// TIA Portal V20 export
FUNCTION_BLOCK "FC_Traffic_Lights"   // FB1, LAD
{ S7_Optimized_Access := 'TRUE' }
// stored: MemoryReserve 100, SetENOAutomatically false
   VAR
      "Timer" { S7_SetPoint := 'True'} : TON_TIME;
   END_VAR
   VAR_TEMP   // added for the SCL form of the ladder/FBD networks
      _w1 : Bool;
   END_VAR
BEGIN

REGION Network 1
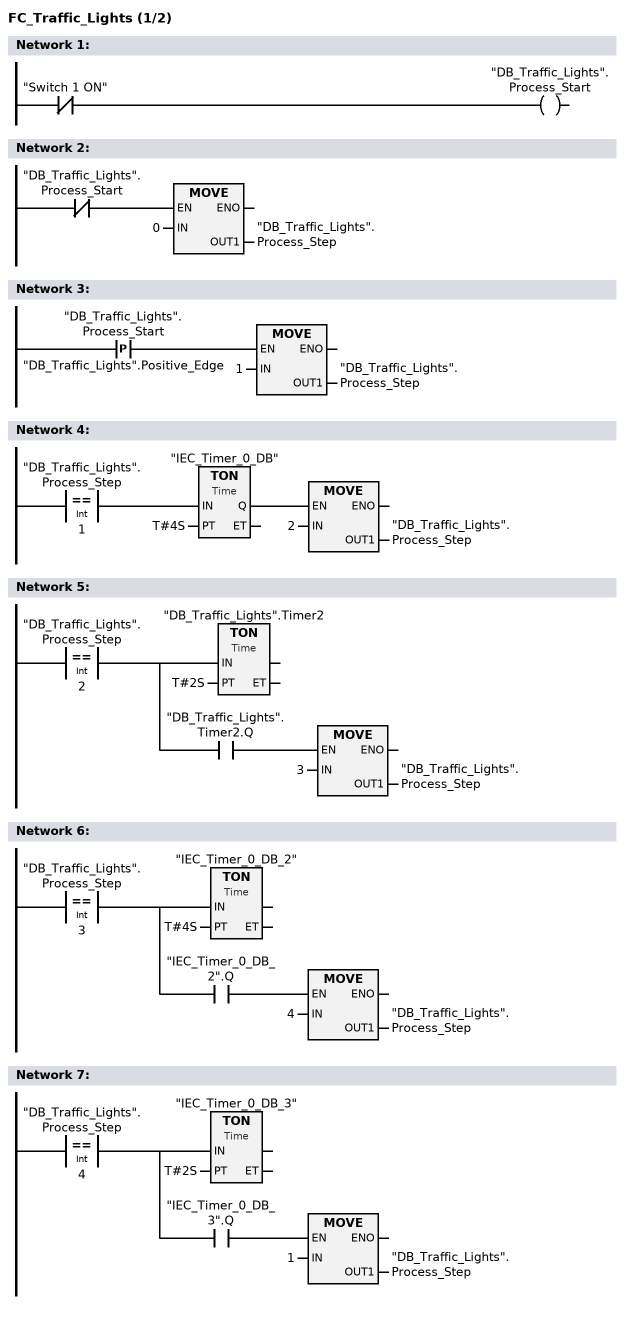
   RUNG wire#powerrail
      I_Contact( "Switch 1 ON" )
      Coil( "DB_Traffic_Lights".Process_Start )
   END_RUNG
   // the same network as SCL:
   "DB_Traffic_Lights".Process_Start := NOT "Switch 1 ON";
END_REGION

REGION Network 2
   RUNG wire#powerrail
      I_Contact( "DB_Traffic_Lights".Process_Start )
      Move(in := 0, out1 => "DB_Traffic_Lights".Process_Step)
   END_RUNG
   // the same network as SCL:
   IF NOT "DB_Traffic_Lights".Process_Start THEN "DB_Traffic_Lights".Process_Step := 0; END_IF;
END_REGION

REGION Network 3
   RUNG wire#powerrail
      P_Contact(operand := "DB_Traffic_Lights".Process_Start, bit := "DB_Traffic_Lights".Positive_Edge)
      Move(in := 1, out1 => "DB_Traffic_Lights".Process_Step)
   END_RUNG
   // the same network as SCL:
   #_w1 := "DB_Traffic_Lights".Process_Start AND NOT "DB_Traffic_Lights".Positive_Edge;   // rising edge of "DB_Traffic_Lights".Process_Start
   "DB_Traffic_Lights".Positive_Edge := "DB_Traffic_Lights".Process_Start;
   IF #_w1 THEN "DB_Traffic_Lights".Process_Step := 1; END_IF;
END_REGION

REGION Network 4
   RUNG wire#powerrail
      { S7_Templates := "SrcType := Int" } EQ_Contact(in1 := "DB_Traffic_Lights".Process_Step, in2 := 1)
      { S7_Templates := "time_type := Time" } "IEC_Timer_0_DB".TON(pt := T#4S, et =>)
      Move(in := 2, out1 => "DB_Traffic_Lights".Process_Step)
   END_RUNG
   // the same network as SCL:
   "IEC_Timer_0_DB".TON(IN := "DB_Traffic_Lights".Process_Step = 1, PT := T#4S);
   IF "IEC_Timer_0_DB".Q THEN "DB_Traffic_Lights".Process_Step := 2; END_IF;
END_REGION

REGION Network 5
   RUNG wire#powerrail
      { S7_Templates := "SrcType := Int" } EQ_Contact(in1 := "DB_Traffic_Lights".Process_Step, in2 := 2)
      wire#w1
      { S7_Templates := "time_type := Time" } "DB_Traffic_Lights".Timer2.TON(pt := T#2S, et =>)
   END_RUNG
   RUNG wire#w1
      Contact( "DB_Traffic_Lights".Timer2.Q )
      Move(in := 3, out1 => "DB_Traffic_Lights".Process_Step)
   END_RUNG
   // the same network as SCL:
   #_w1 := "DB_Traffic_Lights".Process_Step = 2;
   "DB_Traffic_Lights".Timer2.TON(IN := #_w1, PT := T#2S);
   IF #_w1 AND "DB_Traffic_Lights".Timer2.Q THEN "DB_Traffic_Lights".Process_Step := 3; END_IF;
END_REGION

REGION Network 6
   RUNG wire#powerrail
      { S7_Templates := "SrcType := Int" } EQ_Contact(in1 := "DB_Traffic_Lights".Process_Step, in2 := 3)
      wire#w1
      { S7_Templates := "time_type := Time" } "IEC_Timer_0_DB_2".TON(pt := T#4S, et =>)
   END_RUNG
   RUNG wire#w1
      Contact( "IEC_Timer_0_DB_2".Q )
      Move(in := 4, out1 => "DB_Traffic_Lights".Process_Step)
   END_RUNG
   // the same network as SCL:
   #_w1 := "DB_Traffic_Lights".Process_Step = 3;
   "IEC_Timer_0_DB_2".TON(IN := #_w1, PT := T#4S);
   IF #_w1 AND "IEC_Timer_0_DB_2".Q THEN "DB_Traffic_Lights".Process_Step := 4; END_IF;
END_REGION

REGION Network 7
   RUNG wire#powerrail
      { S7_Templates := "SrcType := Int" } EQ_Contact(in1 := "DB_Traffic_Lights".Process_Step, in2 := 4)
      wire#w1
      { S7_Templates := "time_type := Time" } "IEC_Timer_0_DB_3".TON(pt := T#2S, et =>)
   END_RUNG
   RUNG wire#w1
      Contact( "IEC_Timer_0_DB_3".Q )
      Move(in := 1, out1 => "DB_Traffic_Lights".Process_Step)
   END_RUNG
   // the same network as SCL:
   #_w1 := "DB_Traffic_Lights".Process_Step = 4;
   "IEC_Timer_0_DB_3".TON(IN := #_w1, PT := T#2S);
   IF #_w1 AND "IEC_Timer_0_DB_3".Q THEN "DB_Traffic_Lights".Process_Step := 1; END_IF;
END_REGION

REGION Network 8: Step
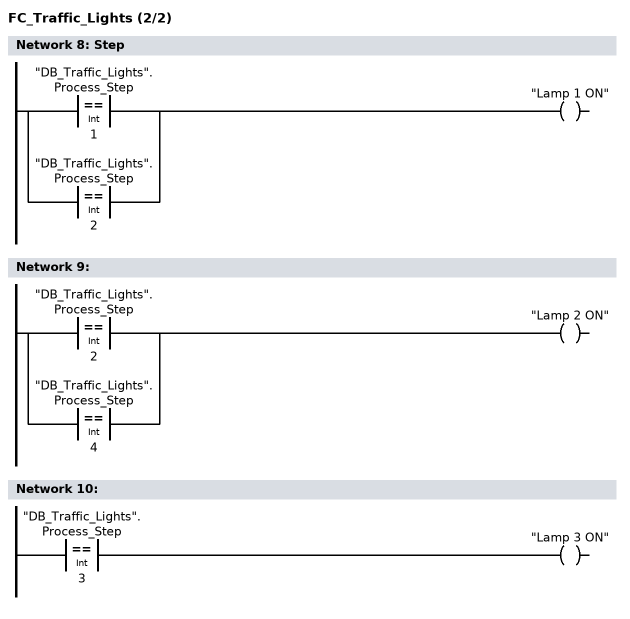
   RUNG wire#powerrail
      { S7_Templates := "SrcType := Int" } EQ_Contact(in1 := "DB_Traffic_Lights".Process_Step, in2 := 1)
      wire#w1
      Coil( "Lamp 1 ON" )
   END_RUNG
   RUNG wire#powerrail
      { S7_Templates := "SrcType := Int" } EQ_Contact(in1 := "DB_Traffic_Lights".Process_Step, in2 := 2)
   END_RUNG wire#w1
   // the same network as SCL:
   "Lamp 1 ON" := ("DB_Traffic_Lights".Process_Step = 1) OR ("DB_Traffic_Lights".Process_Step = 2);
END_REGION

REGION Network 9
   RUNG wire#powerrail
      { S7_Templates := "SrcType := Int" } EQ_Contact(in1 := "DB_Traffic_Lights".Process_Step, in2 := 2)
      wire#w1
      Coil( "Lamp 2 ON" )
   END_RUNG
   RUNG wire#powerrail
      { S7_Templates := "SrcType := Int" } EQ_Contact(in1 := "DB_Traffic_Lights".Process_Step, in2 := 4)
   END_RUNG wire#w1
   // the same network as SCL:
   "Lamp 2 ON" := ("DB_Traffic_Lights".Process_Step = 2) OR ("DB_Traffic_Lights".Process_Step = 4);
END_REGION

REGION Network 10
   RUNG wire#powerrail
      { S7_Templates := "SrcType := Int" } EQ_Contact(in1 := "DB_Traffic_Lights".Process_Step, in2 := 3)
      Coil( "Lamp 3 ON" )
   END_RUNG
   // the same network as SCL:
   "Lamp 3 ON" := "DB_Traffic_Lights".Process_Step = 3;
END_REGION
END_FUNCTION_BLOCK
